FUNCTION FC_Add : WORD
VAR_INPUT
	a :WORD;
	b :WORD;
END_VAR
VAR
END_VAR

FC_Add := a+b;

END_FUNCTION

(* stored: Version 1.1.0.1
   POU FC_Add: Id {681ed6ca-72dc-4e7c-9e20-ed27f3d4f117}, SpecialFunc None *)
